FUNCTION_BLOCK FB_Shutdown IMPLEMENTS I_ShutDown
VAR_INPUT
END_VAR
VAR_OUTPUT
END_VAR
VAR
END_VAR

{warning 'add method implementation '}
METHOD ShutDown : BOOL
VAR_INPUT
	GvlIdentifier	: STRING;
END_VAR
//IF GvlIdentifier = 'R1' THEN
//	R1.RecipeStatus		:= FALSE;
//	R1.HeatCoolStatus	:= FALSE;
//	R1.StirrerStatus	:= FALSE;
//	R1.AbortRecipe		:= FALSE;
//END_IF;
END_METHOD

END_FUNCTION_BLOCK

(* stored: Version 1.1.0.1, ProductVersion 3.1.4024.6
   POU FB_Shutdown: Id {41d600f1-2237-4a02-b3af-e31def017b6b}, SpecialFunc None
   Method ShutDown: Id {fcb05a15-7607-42b3-85e6-d7399a1ca780} *)
